# B&R Automation Studio project Lab_1
Automation Studio 4.5.2.102

## Configuration Config1

CPU 4PP065.0571-P74, AutomationRuntime D4.52, Build 4.1.2, Vc V4.52.0

### Task classes (Cpu.sw)
```
Cyclic#1:
  Program <- Program.prg
DataObjects: Acp10sys
NcDataObjects: acp10etxen <- acp10etxen.dob
Binaries: udbdef, TCData, arconfig, User, sysconf, iomap, asfw, ashwac, ashwd, Role, acp10cfg, Acp10map
Libraries: Acp10man, Acp10par, NcGlobal, Acp10sdc, AsBrStr, powerlnk, astime, fileio, runtime
```

### Hardware
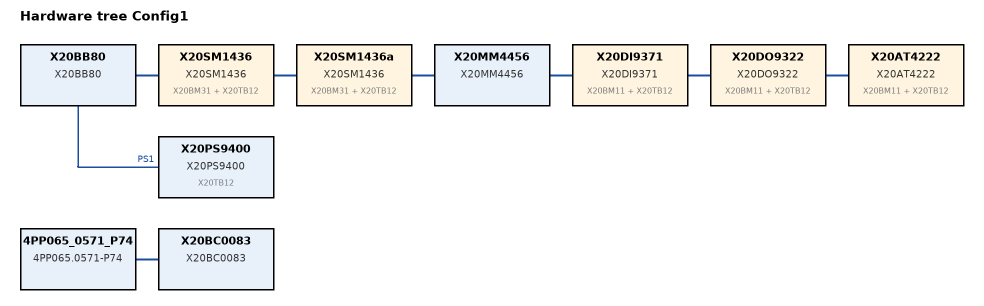
```
4PP065_0571_P74 : 4PP065.0571-P74 v1.1.2.0
  Connector IF5:
    ActivateDevice = 1
    Mode = Manual
    InternetAddress = 127.0.0.1
    SubnetMask = 255.255.255.0
  ConfigurationID = labBR
  Simulation = 1
  TimerDeviceType = EPLX2X
  TimerDevice = 4PP065_0571_P74.IF4
  TaskClassIdleTime = 2000
  Cyclic1Output = 1
X20AT4222 : X20AT4222 v1.2.3.0  [SS1 -> X20TB12e.SS; SL -> X20BM11b.SL1]
X20BB80 : X20BB80 v1.0.2.0
X20BC0083 : X20BC0083 v2.7.0.0  [PLK1 -> 4PP065_0571_P74.IF4 [Cable Type=PowerlinkCable, Length=10, Version=1.0.0.2]; SL -> X20BB80.SL1]
X20BM11 : X20BM11 v1.0.0.1  [X2X1 -> X20MM4456.X2X2]
X20BM11a : X20BM11 v1.0.0.1  [X2X1 -> X20BM11.X2X2]
X20BM11b : X20BM11 v1.0.0.1  [X2X1 -> X20BM11a.X2X2]
X20BM31 : X20BM31 v1.0.0.1  [X2X1 -> X20BB80.IF1]
X20BM31a : X20BM31 v1.0.0.1  [X2X1 -> X20BM31.X2X2]
X20DI9371 : X20DI9371 v1.0.2.0  [SS1 -> X20TB12c.SS; SL -> X20BM11.SL1]
X20DO9322 : X20DO9322 v1.0.3.0  [SS1 -> X20TB12d.SS; SL -> X20BM11a.SL1]
X20MM4456 : X20MM4456 v1.1.5.0  [X2X1 -> X20BM31a.X2X2]
X20PS9400 : X20PS9400 v1.0.2.4  [SS1 -> X20TB12.SS; PS -> X20BB80.PS1]
X20SM1436 : X20SM1436 v1.4.2.1  [SS1 -> X20TB12a.SS; SL -> X20BM31.SL1]
X20SM1436a : X20SM1436 v1.4.2.1  [SS1 -> X20TB12b.SS; SL -> X20BM31a.SL1]
X20TB12 : X20TB12 v1.0.0.0
X20TB12a : X20TB12 v1.0.0.0
X20TB12b : X20TB12 v1.0.0.0
X20TB12c : X20TB12 v1.0.0.0
X20TB12d : X20TB12 v1.0.0.0
X20TB12e : X20TB12 v1.0.0.0
```

### IoMap.iom - 4PP065_0571_P74/IoMap.iom
```iecst
VAR_CONFIG
	::Program:Led1 AT %QX."X20DO9322".DigitalOutput02;
	::Program:Led2 AT %QX."X20DO9322".DigitalOutput03;
	::Program:Led3 AT %QX."X20DO9322".DigitalOutput04;
	::Program:Led4 AT %QX."X20DO9322".DigitalOutput05;
END_VAR
```

### Acp10map.ncm - 4PP065_0571_P74/Motion/Acp10map.ncm
```
NcMapping (NcSwId=Acp10)
  NcObject X20SM1436a_ncAXIS1 (ModuleId=X20SM1436a, ModuleAddress=SDC_IF1.ST1, Type=ncAXIS, Channel=1, AcoposSimulation=Off, Disabled=TRUE, ModuleDisabled=FALSE)
  NcObject X20SM1436_ncAXIS1 (ModuleId=X20SM1436, ModuleAddress=SDC_IF1.ST2, Type=ncAXIS, Channel=1, AcoposSimulation=Off, Disabled=TRUE, ModuleDisabled=FALSE)
```

## Logical view

### Program Logical/Program

#### Variables.var
```iecst
VAR
	Led1 : BOOL;
	Led2 : BOOL;
	Led3 : BOOL;
	Led4 : BOOL;
	Counter : USINT;
END_VAR
```

#### Main.c
```c
#include <bur/plctypes.h>

#ifdef _DEFAULT_INCLUDES
	#include <AsDefault.h>
#endif

void _INIT ProgramInit(void) {

}

void _CYCLIC ProgramCyclic(void) {
	if (Counter % 2) {
		Led1 = !Led1;
	}
	if (Counter % 5) {
		Led2 = !Led2;
	}
	if (Counter % 10) {
		Led3 = !Led3;
	}
	if (Counter % 20) {
		Led4 = !Led4;
	}
	Counter++;
}

void _EXIT ProgramExit(void) {

}
```
